(*
SPDX-FileCopyrightText: © 2026 Oleksandr Tiutyk <trofimich@gmail.com>
SPDX-License-Identifier: MIT
License: https://opensource.org/license/mit
*)

INTERFACE IVariableContainer EXTENDS TOF_Core.IObject

METHOD TryGetVariable : BOOL
VAR_INPUT
	name : STRING;
END_VAR
VAR_OUTPUT
	variable : TOF_Core.GENERIC_VALUE;
END_VAR
END_METHOD

END_INTERFACE

(* stored: Version 1.1.0.1
   Itf IVariableContainer: Id {a821d865-7499-4823-bc9c-a9226b7ccd87}
   Method TryGetVariable: Id {cde7c073-74e9-49f1-ac46-4fe75c6c0e26} *)
